TYPE CResult :
STRUCT
	datatype	: INT;
	result		: BOOL;
END_STRUCT
END_TYPE

(* stored: Version 1.1.0.1, ProductVersion 3.1.4024.11
   DUT CResult: Id {665fdde3-d1a8-4d7c-853c-844994aded07} *)
